TYPE "UDT_Chiller_Raw"
VERSION : 0.1
   STRUCT
      IN_OutletTemp : Int;   // Outlet Temperature
      IN_InletTemp : Int;    // Inlet Temperature
   END_STRUCT;

END_TYPE

TYPE "UDT_Chiller_Data"
VERSION : 0.1
   STRUCT
      OUT_Heartbeat : Int;    // Heartbeat Signal
      OUT_OutletTemp : Real;  // Outlet Temperature
      OUT_InletTemp : Real;   // Inlet Temperature
   END_STRUCT;

END_TYPE